FUNCTION_BLOCK centralTwoConCtl2 (* Composite Function Block Type *)
  (* Standard: 61499-2 *)
  (* Version 0.2, 2003-12-05, JHC, Rockwell Automation, Renamed from NEWCOMPFB. *)
  (* Version 0.1, 2002-01-08, JHC, Rockwell Automation, Added DLY FB as example. *)
  (* Version 0.0, 2000-05-27, JHC, Rockwell Automation *)
  (* Compiler header: package fb.rt.cs725; *)
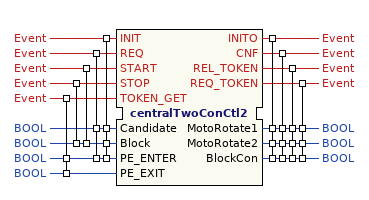
  EVENT_INPUT
    INIT WITH Candidate, Block, PE_ENTER; (* Initialization Request *)
    REQ WITH Candidate, PE_ENTER; (* Normal Execution Request *)
    START WITH Block;
    STOP WITH Block;
    TOKEN_GET WITH PE_EXIT, PE_ENTER;
  END_EVENT
  EVENT_OUTPUT
    INITO WITH MotoRotate1, MotoRotate2, BlockCon; (* Initialization Confirm *)
    CNF WITH MotoRotate1, MotoRotate2, BlockCon; (* Execution Confirmation *)
    REL_TOKEN WITH MotoRotate1, MotoRotate2, BlockCon;
    REQ_TOKEN WITH MotoRotate1, MotoRotate2, BlockCon;
  END_EVENT
  VAR_INPUT
    Candidate : BOOL;
    Block : BOOL;
    PE_ENTER : BOOL;
    PE_EXIT : BOOL;
  END_VAR
  VAR_OUTPUT
    MotoRotate1 : BOOL;
    MotoRotate2 : BOOL;
    BlockCon : BOOL;
  END_VAR
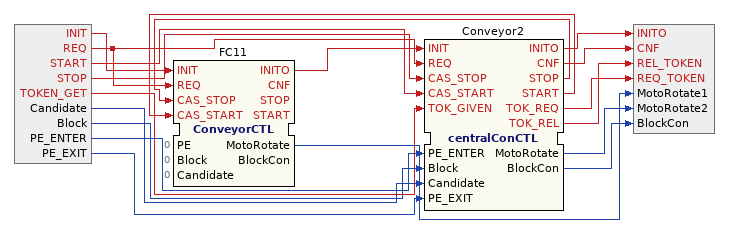
  FBS
    FC11 : ConveyorCTL(PE := 0, Block := 0, Candidate := 0);
    Conveyor2 : centralConCTL;
  END_FBS
  EVENT_CONNECTIONS
    INIT TO FC11.INIT;
    REQ TO FC11.REQ;
    FC11.INITO TO Conveyor2.INIT;
    REQ TO Conveyor2.REQ;
    STOP TO Conveyor2.CAS_STOP;
    START TO Conveyor2.CAS_START;
    TOKEN_GET TO Conveyor2.TOK_GIVEN;
    Conveyor2.INITO TO INITO;
    Conveyor2.CNF TO CNF;
    Conveyor2.TOK_REQ TO REQ_TOKEN;
    Conveyor2.TOK_REL TO REL_TOKEN;
    Conveyor2.STOP TO FC11.CAS_STOP;
    Conveyor2.START TO FC11.CAS_START;
  END_CONNECTIONS
  DATA_CONNECTIONS
    FC11.MotoRotate TO MotoRotate1;
    PE_ENTER TO Conveyor2.PE_ENTER;
    Block TO Conveyor2.Block;
    Candidate TO Conveyor2.Candidate;
    PE_EXIT TO Conveyor2.PE_EXIT;
    Conveyor2.MotoRotate TO MotoRotate2;
    Conveyor2.BlockCon TO BlockCon;
  END_CONNECTIONS
END_FUNCTION_BLOCK
